// TIA Portal V20 export
FUNCTION_BLOCK "MotorGroups"   // FB3, LAD
{ S7_Optimized_Access := 'TRUE' }
// stored: AutoNumber false
   VAR
      Group1 { S7_SetPoint := 'True'} : "MotorSequenceLAD";
      Group2 { S7_SetPoint := 'True'} : "MotorSequenceLAD";
   END_VAR
BEGIN

REGION Network 1
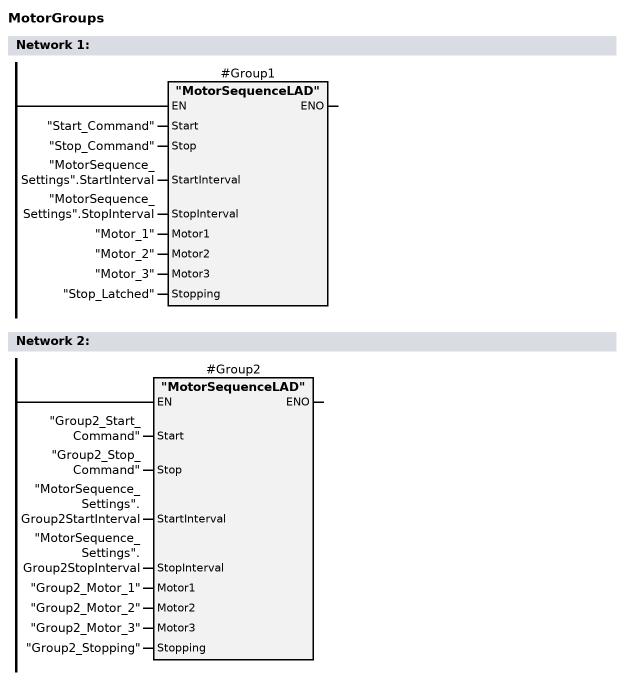
   RUNG wire#powerrail
      #Group1(Start := "Start_Command", Stop := "Stop_Command", StartInterval := "MotorSequence_Settings".StartInterval, StopInterval := "MotorSequence_Settings".StopInterval, Motor1 := "Motor_1", Motor2 := "Motor_2", Motor3 := "Motor_3", Stopping := "Stop_Latched")
   END_RUNG
   // the same network as SCL:
   #Group1(Start := "Start_Command",   // "MotorSequenceLAD"
           Stop := "Stop_Command",
           StartInterval := "MotorSequence_Settings".StartInterval,
           StopInterval := "MotorSequence_Settings".StopInterval,
           Motor1 := "Motor_1",
           Motor2 := "Motor_2",
           Motor3 := "Motor_3",
           Stopping := "Stop_Latched");
END_REGION

REGION Network 2
   RUNG wire#powerrail
      #Group2(Start := "Group2_Start_Command", Stop := "Group2_Stop_Command", StartInterval := "MotorSequence_Settings".Group2StartInterval, StopInterval := "MotorSequence_Settings".Group2StopInterval, Motor1 := "Group2_Motor_1", Motor2 := "Group2_Motor_2", Motor3 := "Group2_Motor_3", Stopping := "Group2_Stopping")
   END_RUNG
   // the same network as SCL:
   #Group2(Start := "Group2_Start_Command",   // "MotorSequenceLAD"
           Stop := "Group2_Stop_Command",
           StartInterval := "MotorSequence_Settings".Group2StartInterval,
           StopInterval := "MotorSequence_Settings".Group2StopInterval,
           Motor1 := "Group2_Motor_1",
           Motor2 := "Group2_Motor_2",
           Motor3 := "Group2_Motor_3",
           Stopping := "Group2_Stopping");
END_REGION
END_FUNCTION_BLOCK
